// TIA Portal V16 export
// export: Created 2024-12-03T15:41:42.6190391Z, ExportSetting WithDefaults, DisplayName Totally Integrated Automation Portal, DisplayVersion V16 Update 6, DisplayName TIA Portal Version Control Interface, DisplayVersion V16 Update 2, DisplayName TIA Portal Openness, DisplayVersion V16 Update 6, DisplayName TIA Portal Teamcenter Gateway, DisplayVersion V16, DisplayName SINAMICS Startdrive Advanced, DisplayVersion V16 Update 5, DisplayName SINAMICS Startdrive G130, G150, S120, S150, SINAMICS MV, S210, DisplayVersion V16 Update 5, DisplayName SINAMICS Startdrive G110M, G120, G120C, G120D, G120P, G115D, DisplayVersion V16 Update 5, DisplayName STEP 7 Professional, DisplayVersion V16 Update 6, DisplayName STEP 7 Safety, DisplayVersion V16, DisplayName WinCC Advanced / Unified PC, DisplayVersion V16 Update 6
FUNCTION_BLOCK "G120DPosControl_FB"   // FB49, SCL
{ S7_Optimized_Access := 'TRUE' }
VERSION : 0.1
// stored: AutoNumber true, IsIECCheckEnabled false, IsRetainMemResEnabled false, MemoryReserve 100, SetENOAutomatically false, UDAEnableTagReadback false
   VAR_INPUT
      I_HWIDSTW : HW_IO;
      I_HWIDZSW : HW_IO;
      I_Home : Bool;
      I_Interlock : Bool;
      I_SafetyProx_1 : Bool;
      I_SafetyProx_2 : Bool;
      I_ExtReset : Bool := true;
   END_VAR
   VAR_IN_OUT
      IO_DRIVE : "G120D_SINAPOS_UDT";
   END_VAR
   VAR
      cycle : "CycleRun";
      alarm { S7_SetPoint := 'True'} : "AlarmInfo_UDT";
      reset { S7_SetPoint := 'True'} : TOF_TIME;
      disconnected { S7_SetPoint := 'True'} : TON_TIME;
      notOn { S7_SetPoint := 'True'} : TON_TIME;
      notEnabled { S7_SetPoint := 'True'} : TON_TIME;
      EposConfig { S7_SetPoint := 'True'} : DWord;
      controller : SinaPos;
      jog_1 { S7_SetPoint := 'True'} : "HeartBeatButton_FB";
      jog_2 { S7_SetPoint := 'True'} : "HeartBeatButton_FB";
      homed { S7_SetPoint := 'True'} : Bool;
      homeStep : DInt;
      AlarmActive : Program_Alarm;
      NotHomed : Program_Alarm;
      FaultActive : Program_Alarm;
      FaultDisconnected : Program_Alarm;
      FaultNotOnTimedOut : Program_Alarm;
      FaultNotReady : Program_Alarm;
      SafetyProx_1 : Program_Alarm;
      SafetyProx_2 : Program_Alarm;
      FaultSafetyError : Program_Alarm;
      FaultSto : Program_Alarm;
   END_VAR
   VAR_TEMP
      T_Appstate : "ApplicationState_UDT";
      T_Zone : "ZoneInfo";
      T_Mode : Int;
      T_On : Bool;
      T_Direction : Bool;
      T_Reset : Bool;
      T_ExecuteMode : Bool;
      T_Position : DInt;
      T_Speed : DInt;
      T_Condition : Bool;
   END_VAR
BEGIN
   REGION APPSTATE

       #T_Zone := "ApplicationState_DB".ZoneNames[#IO_DRIVE.Zone];
       #T_Appstate := "ApplicationState_DB".Appstate[#T_Zone.AppStateIndex];

   END_REGION

   REGION COMMANDS

       //Always reset
       #T_Mode := 0;
       #T_On := 0;
       #T_Direction := 0;
       #T_ExecuteMode := 0;
       #T_Position := 0;
       #T_Speed := 0;


       REGION AUTO

           IF #T_Appstate.States.AutoModeActivated.State AND #IO_DRIVE.Status.homed THEN
               #T_Mode := #IO_DRIVE.Cmd.auto.mode;
               #T_On := #IO_DRIVE.Cmd.auto.enable;
               #T_Direction := #IO_DRIVE.Cmd.auto.direction;
               #T_ExecuteMode := #IO_DRIVE.Cmd.auto.executeMode;
               #T_Position := REAL_TO_DINT(#IO_DRIVE.Cmd.auto.pos);
               #T_Speed := REAL_TO_DINT(IN := #IO_DRIVE.Cmd.auto.speed);

               REGION set speed

                   #IO_DRIVE.Settings.VelocityOverride := 100;
                   #IO_DRIVE.Settings.AccelerationOverride := 100;
                   #IO_DRIVE.Settings.DeaccelarationOverride := 100;

               END_REGION

           END_IF;

       END_REGION

       REGION MANUAL

           "Util_HandShaked_FC"(#IO_DRIVE.Cmd.manual.stop);

           #jog_1(IO_Beat:=#IO_DRIVE.Cmd.manual.jog1);
           #jog_2(IO_Beat := #IO_DRIVE.Cmd.manual.jog2);

           REGION JOGGING

               #IO_DRIVE.Cmd.manual.jog1.state := #IO_DRIVE.Cmd.manual.jog1.state AND NOT #IO_DRIVE.Faults.SafetyProx_1;
               #IO_DRIVE.Cmd.manual.jog2.state := #IO_DRIVE.Cmd.manual.jog2.state AND NOT #IO_DRIVE.Faults.SafetyProx_2;


               IF #T_Appstate.States.ManualModeActivated.State AND NOT #IO_DRIVE.Cmd.manual.activateHoming THEN
                   #T_Mode := 7;
                   #T_On := #IO_DRIVE.Cmd.manual.jog1.state OR #IO_DRIVE.Cmd.manual.jog2.state;
                   #T_Direction := #IO_DRIVE.Cmd.manual.jog2.state;

                   REGION set speed

                       #IO_DRIVE.Settings.VelocityOverride := REAL_TO_INT(#IO_DRIVE.Cmd.manual.speed);

                       IF #IO_DRIVE.Settings.VelocityOverride > #IO_DRIVE.Settings.maxJogSpeed THEN
                           #IO_DRIVE.Settings.VelocityOverride := #IO_DRIVE.Settings.maxJogSpeed;
                       END_IF;

                       IF #IO_DRIVE.Settings.VelocityOverride < #IO_DRIVE.Settings.minJogSpeed THEN
                           #IO_DRIVE.Settings.VelocityOverride := #IO_DRIVE.Settings.minJogSpeed;
                       END_IF;

                       #IO_DRIVE.Settings.AccelerationOverride := 50;
                       #IO_DRIVE.Settings.DeaccelarationOverride := 50;

                   END_REGION

               END_IF;

           END_REGION

           REGION HOMING

               IF #IO_DRIVE.Faults.SafetyProx_1 OR #IO_DRIVE.Faults.SafetyProx_2 THEN
                   #homed := 0;
               END_IF;

               #IO_DRIVE.Status.homed := #homed AND #controller.AxisRef;

               REGION HOME SEQUENCE

                   IF #IO_DRIVE.Cmd.manual.stop.signal THEN
                       #IO_DRIVE.Cmd.manual.activateHoming := 0;
                   END_IF;

                   IF #T_Appstate.States.ManualModeActivated.State AND #IO_DRIVE.Cmd.manual.activateHoming THEN
                       #T_Mode := 4;
                       #T_On := 1;
                       #T_ExecuteMode := #IO_DRIVE.Status.enabled AND #IO_DRIVE.Status.CurrentMode = 4;
                       #T_Speed := 1000;
                       #IO_DRIVE.Settings.VelocityOverride := 100;
                       #IO_DRIVE.Settings.AccelerationOverride := 50;
                       #IO_DRIVE.Settings.DeaccelarationOverride := 50;
                   END_IF;

                   IF #IO_DRIVE.Status.CurrentMode = 4 AND #IO_DRIVE.Status.homed THEN
                       #IO_DRIVE.Cmd.manual.activateHoming := 0;
                   END_IF;

               END_REGION

           END_REGION

           IF NOT #T_Appstate.States.ManualModeActivated.State THEN
               #IO_DRIVE.Cmd.manual.activateHoming := 0;
               #IO_DRIVE.Cmd.manual.jog1.beat := 0;
               #IO_DRIVE.Cmd.manual.jog2.beat := 0;
               #IO_DRIVE.Cmd.manual.speed := 0;
               #IO_DRIVE.Cmd.manual.stop.signal := 0;
           END_IF;
       END_REGION

       REGION RESET COMMAND ON ERROR 
           // then we don't start after reset :)

           REGION INTERLOCK ON AUTO
               IF #T_Appstate.States.AutoModeActivated.State AND
                   (#IO_DRIVE.Faults.status > 0 OR NOT #T_Appstate.States.EmergencyOk.State OR #I_Interlock) THEN

                   #T_On := 0;
                   #T_Direction := 0;
                   #T_ExecuteMode := 0;
                   #T_Speed := 0;

               END_IF;
           END_REGION

           REGION INTERLOCK ON MANUAL

               #T_Condition :=
               #IO_DRIVE.Faults.Disconnected OR
               #IO_DRIVE.Faults.FaultActive OR
               #IO_DRIVE.Faults.NotOnTImedOut OR
               #IO_DRIVE.Faults.NotReady;


               #T_Condition := #T_Condition OR
               ((#IO_DRIVE.Faults.SafetyProx_1 OR #IO_DRIVE.Faults.SafetyProx_2) AND #T_Mode = 4); //Homing

               #T_Condition := #T_Condition OR #I_Interlock;

               IF #T_Appstate.States.ManualModeActivated.State AND
                   (#T_Condition OR NOT #T_Appstate.States.EmergencyOk.State) THEN

                   #IO_DRIVE.Cmd.manual.activateHoming := 0;
                   #T_Mode := 0;
                   #T_On := 0;
                   #T_Direction := 0;
                   #T_ExecuteMode := 0;
                   #T_Speed := 0;

               END_IF;

           END_REGION

       END_REGION

   END_REGION

   REGION SINA POS CONTROLLER

       #EposConfig.%X0 := 1;
       #EposConfig.%X1 := 1;
       #EposConfig.%X6 := #I_Home;
       #EposConfig.%X8 := 1;

                   #controller(ModePos:=#T_Mode,
                   EnableAxis:=#T_On,
                   CancelTraversing:=TRUE,
                   IntermediateStop:=#T_Appstate.States.EmergencyOk.State,
                   Positive:=NOT #T_Direction,
                   Negative:=#T_Direction,
                   Jog1:=#T_On AND NOT #T_Direction AND #T_Mode = 7,
                   Jog2:=#T_On AND #T_Direction AND #T_Mode = 7 ,
                   FlyRef:=FALSE,
                   ExecuteMode:=#T_ExecuteMode,
                   Position:=#T_Position,
                   Velocity:=#T_Speed,
                   OverV:=#IO_DRIVE.Settings.VelocityOverride,
                   OverAcc := #IO_DRIVE.Settings.AccelerationOverride,
                   OverDec := #IO_DRIVE.Settings.DeaccelarationOverride,
                   ConfigEPos:=#EposConfig,
                   HWIDSTW:=#I_HWIDSTW,
                   HWIDZSW:=#I_HWIDZSW,
                   AxisEnabled=>#IO_DRIVE.Status.enabled,
                   AxisPosOk=>#IO_DRIVE.Status.atPosition,
                   Lockout=>#IO_DRIVE.Status.Running,
                   ActMode=>#IO_DRIVE.Status.CurrentMode);

       #IO_DRIVE.Status.ActualSpeed := DINT_TO_REAL(IN := #controller.ActVelocity);
       #IO_DRIVE.Status.ActualPosition := DINT_TO_REAL(IN := #controller.ActPosition);

   END_REGION

   REGION CYCLE COUNTER

       IF "GlobalCycleRunner_FB_DB".O_Cycle = #T_Zone.AppStateIndex THEN
           #cycle();
       END_IF;

   END_REGION

   REGION STATUS

       #IO_DRIVE.Status.ActualDirection := #IO_DRIVE.Status.ActualSpeed < 0.0;
       #IO_DRIVE.Status.Running := #IO_DRIVE.Status.ActualSpeed <> 0.0;

       #IO_DRIVE.Status.CmdRunManualActive := #T_On AND #IO_DRIVE.Status.ManualModeActive;

       //#IO_DRIVE.Status.Interlocked := #IO_DRIVE.Cmd.Interlock;

       #IO_DRIVE.Status.ManualCommandsDisabled := TRUE;
       #IO_DRIVE.Status.ManualModeActive := #T_Appstate.States.ManualModeActivated.State;

   END_REGION

   REGION ALARM / FAULT INFO

       IF NOT #alarm.init OR #IO_DRIVE.info.Name = '' THEN
           #IO_DRIVE.info.Name := "buildObjectName"(I_Symbolname := GetSymbolName(variable := #IO_DRIVE, size := 100));
           #alarm.info := "buildAlarmInfo"(I_ObjectName := #IO_DRIVE.info.Name, I_ZoneIndex := #IO_DRIVE.Zone, I_ZoneName := #T_Zone.ZoneName);
           #alarm.init := true;
       END_IF;

   END_REGION

   REGION ALARMS

       #IO_DRIVE.Alarms.AlarmCode := #controller.ActWarn;

       REGION ALARM FROM DRIVE X0

           #IO_DRIVE.Alarms.AlarmFromDrive := #controller.Error;
           #IO_DRIVE.Alarms.Status.%X0 := #IO_DRIVE.Alarms.AlarmFromDrive;

       END_REGION

       REGION NOT HOMED X1

           #IO_DRIVE.Alarms.NotHomed := NOT #IO_DRIVE.Status.homed;
           #IO_DRIVE.Alarms.Status.%X1 := #IO_DRIVE.Alarms.NotHomed;

           #NotHomed(SIG := #IO_DRIVE.Alarms.NotHomed,
                     SD_1 := #alarm.info,
                     SD_2 := #T_Zone.ZoneName,
                     SD_3 := #IO_DRIVE.info.Name);

       END_REGION

       REGION PROGRAM ALARMS

           IF "GlobalCycleRunner_FB_DB".O_Cycle = #T_Zone.AppStateIndex AND #cycle.O_Cycle = 1 THEN

               #AlarmActive(SIG := #IO_DRIVE.Alarms.AlarmFromDrive,
                                SD_1 := #alarm.info,
                                SD_2 := #T_Zone.ZoneName,
                                SD_3 := #IO_DRIVE.info.Name,
                                SD_4 := #IO_DRIVE.Alarms.AlarmCode);

           END_IF;

       END_REGION

       REGION ALARM ACTIVE

           IF #IO_DRIVE.Alarms.Status > 0 THEN
               "ApplicationState_DB".Appstate[#T_Zone.AppStateIndex].Alarms.AlarmActiveInternalPLC := 1;
           END_IF;

       END_REGION

   END_REGION

   REGION FAULTS

       #IO_DRIVE.Faults.FaultCode := #controller.ActFault;

       REGION X0 - FAULT ACTIVE

           IF #IO_DRIVE.Faults.FaultCode > 0 THEN
               #IO_DRIVE.Faults.FaultActive := 1;
           END_IF;

           #IO_DRIVE.Faults.status.%X0 := #IO_DRIVE.Faults.FaultActive;

       END_REGION

       REGION X1 - DISCONNECTED

           #disconnected(IN := #controller.Status = 16#8600 OR #controller.Status = 16#8601,
                         PT := t#500ms);

           IF #disconnected.Q THEN
               #IO_DRIVE.Faults.Disconnected := 1;
           END_IF;

           #IO_DRIVE.Faults.status.%X1 := #IO_DRIVE.Faults.Disconnected;

       END_REGION

       REGION X3 - NOT ON TIMED OUT

           #notOn(IN := NOT #IO_DRIVE.Status.Running AND #T_On AND #IO_DRIVE.Status.CurrentMode = 7,
                  PT := t#500ms);

           IF #notOn.Q THEN
               #IO_DRIVE.Faults.NotOnTImedOut := 1;
           END_IF;

           #IO_DRIVE.Faults.status.%X3 := #IO_DRIVE.Faults.NotOnTImedOut;

       END_REGION

       REGION X4 - NOT READY

           #notEnabled(IN := NOT #IO_DRIVE.Status.enabled AND #IO_DRIVE.Status.CurrentMode > 0 AND #T_On,
      PT := t#500ms);


           IF #notEnabled.Q THEN
               #IO_DRIVE.Faults.NotReady := 1;
           END_IF;

           #IO_DRIVE.Faults.status.%X4 := #IO_DRIVE.Faults.NotReady;

       END_REGION

       REGION X5 - SAFETY PROX 1

           IF #I_SafetyProx_1 THEN
               #IO_DRIVE.Faults.SafetyProx_1 := 1;
           END_IF;

           #IO_DRIVE.Faults.status.%X5 := #IO_DRIVE.Faults.SafetyProx_1;

       END_REGION

       REGION X6 - SAFETY PROX 2

           IF #I_SafetyProx_2 THEN
               #IO_DRIVE.Faults.SafetyProx_2 := 1;
           END_IF;

           #IO_DRIVE.Faults.status.%X6 := #IO_DRIVE.Faults.SafetyProx_2;

       END_REGION

       REGION X7 - SAFETY ERROR

           #IO_DRIVE.Faults.status.%X7 := #IO_DRIVE.Faults.SAFETY_FAULT_ACTIVE;

       END_REGION

       REGION X8 - STO ACTIVE

           #IO_DRIVE.Faults.status.%X8 := #IO_DRIVE.Faults.STO_ACTIVE;

       END_REGION

       REGION PROGRAM ALARM

           IF "GlobalCycleRunner_FB_DB".O_Cycle = #T_Zone.AppStateIndex AND #cycle.O_Cycle = 1 THEN

               #FaultActive(SIG := #IO_DRIVE.Faults.FaultActive,
                            SD_1 := #alarm.info,
                            SD_2 := #T_Zone.ZoneName,
                            SD_3 := #IO_DRIVE.info.Name,
                            SD_4 := #IO_DRIVE.Faults.FaultCode);

           END_IF;

           IF "GlobalCycleRunner_FB_DB".O_Cycle = #T_Zone.AppStateIndex AND #cycle.O_Cycle = 2 THEN

               #FaultDisconnected(SIG := #IO_DRIVE.Faults.Disconnected,
                            SD_1 := #alarm.info,
                            SD_2 := #T_Zone.ZoneName,
                            SD_3 := #IO_DRIVE.info.Name);

           END_IF;

           IF "GlobalCycleRunner_FB_DB".O_Cycle = #T_Zone.AppStateIndex AND #cycle.O_Cycle = 3 THEN

               #FaultNotOnTimedOut(SIG := #IO_DRIVE.Faults.NotOnTImedOut,
                                   SD_1 := #alarm.info,
                                   SD_2 := #T_Zone.ZoneName,
                                   SD_3 := #IO_DRIVE.info.Name);

           END_IF;

           IF "GlobalCycleRunner_FB_DB".O_Cycle = #T_Zone.AppStateIndex AND #cycle.O_Cycle = 4 THEN

               #FaultNotReady(SIG := #IO_DRIVE.Faults.NotReady,
                              SD_1 := #alarm.info,
                              SD_2 := #T_Zone.ZoneName,
                              SD_3 := #IO_DRIVE.info.Name);

           END_IF;

           IF "GlobalCycleRunner_FB_DB".O_Cycle = #T_Zone.AppStateIndex AND #cycle.O_Cycle = 5 THEN

               #SafetyProx_1(SIG := #IO_DRIVE.Faults.SafetyProx_1,
                              SD_1 := #alarm.info,
                              SD_2 := #T_Zone.ZoneName,
                              SD_3 := #IO_DRIVE.info.Name);

           END_IF;

           IF "GlobalCycleRunner_FB_DB".O_Cycle = #T_Zone.AppStateIndex AND #cycle.O_Cycle = 6 THEN

               #SafetyProx_2(SIG := #IO_DRIVE.Faults.SafetyProx_2,
                              SD_1 := #alarm.info,
                              SD_2 := #T_Zone.ZoneName,
                              SD_3 := #IO_DRIVE.info.Name);

            END_IF;

            IF "GlobalCycleRunner_FB_DB".O_Cycle = #T_Zone.AppStateIndex AND #cycle.O_Cycle = 6 THEN

                #FaultSafetyError(SIG := #IO_DRIVE.Faults.SAFETY_FAULT_ACTIVE,
                                  SD_1 := #alarm.info,
                                  SD_2 := #T_Zone.ZoneName,
                                  SD_3 := #IO_DRIVE.info.Name);

            END_IF;

            IF "GlobalCycleRunner_FB_DB".O_Cycle = #T_Zone.AppStateIndex AND #cycle.O_Cycle = 7 THEN

                #FaultSto(SIG := #IO_DRIVE.Faults.STO_ACTIVE,
                          SD_1 := #alarm.info,
                          SD_2 := #T_Zone.ZoneName,
                          SD_3 := #IO_DRIVE.info.Name);

            END_IF;

       END_REGION

       REGION RESET

           #T_Reset := #IO_DRIVE.Cmd.Reset OR (#T_Appstate.Hmi_Buttons.reset.state.LE AND #I_ExtReset);

           #reset(IN := #T_Reset,
                  PT := t#250ms);

           #controller.AckError := 0;
           IF #reset.Q THEN
               #IO_DRIVE.Cmd.Reset := 0;
               #controller.AckError := 1;

               //Reset faults
               #IO_DRIVE.Faults.FaultActive := 0;
               #IO_DRIVE.Faults.Disconnected := 0;
               #IO_DRIVE.Faults.NotOnTImedOut := 0;
               #IO_DRIVE.Faults.NotReady := 0;
               #IO_DRIVE.Faults.SafetyProx_1 := 0;
               #IO_DRIVE.Faults.SafetyProx_2 := 0;

           END_IF;

       END_REGION

       REGION FAULT ACTIVE

           IF #IO_DRIVE.Faults.status > 0 THEN
               "ApplicationState_DB".Appstate[#T_Zone.AppStateIndex].Alarms.AlarmActiveInternalPLC := 1;
           END_IF;

       END_REGION

   END_REGION
END_FUNCTION_BLOCK
